(* IEC 61131-3 sources: com.logicals.lc3.webinar/usRTS_RPMControl_iSOC/src_FB_LIB_SAFE/Convert/LINT, 6 files *)

(* ---- wTRUNC_LINT_TO_DINT.iecst ---- *)
NAMESPACE logicals.web.standard
NAMESPACE convert

/*
 * Function block wrapper for IEC 61131-3 TO_DINT<br>
 * IN =  input value (LINT)<br>
 * OUT = IN (DINT)<br>
 */
FUNCTION_BLOCK wTRUNC_LINT_TO_DINT
	{ vNameAlignment:="center"; altName:="TRUNC_LINT_TO_DINT"; bgColor:="LightPink"; width:=180; hideIONames; }
	VAR_INPUT
		IN : LINT;
	END_VAR
	VAR_OUTPUT
		OUT: DINT;
	END_VAR

	OUT := TO_DINT(IN:=IN, ENO=>ENO);
END_FUNCTION_BLOCK

END_NAMESPACE
END_NAMESPACE

(* ---- wTRUNC_LINT_TO_INT.iecst ---- *)
NAMESPACE logicals.web.standard
NAMESPACE convert

/*
 * Function block wrapper for IEC 61131-3 TO_INT<br>
 * IN =  input value (LINT)<br>
 * OUT = IN (INT)<br>
 */
FUNCTION_BLOCK wTRUNC_LINT_TO_INT
	{ vNameAlignment:="center"; altName:="TRUNC_LINT_TO_INT"; bgColor:="LightPink"; width:=180; hideIONames; }
	VAR_INPUT
		IN : LINT;
	END_VAR
	VAR_OUTPUT
		OUT: INT;
	END_VAR

	OUT := TO_INT(IN:=IN, ENO=>ENO);
END_FUNCTION_BLOCK

END_NAMESPACE
END_NAMESPACE

(* ---- wTRUNC_LINT_TO_LREAL.iecst ---- *)
NAMESPACE logicals.web.standard
NAMESPACE convert

/*
 * Function block wrapper for IEC 61131-3 TO_LREAL<br>
 * IN =  input value (LINT)<br>
 * OUT = IN (LREAL)<br>
 */
FUNCTION_BLOCK wTRUNC_LINT_TO_LREAL
	{ vNameAlignment:="center"; altName:="TRUNC_LINT_TO_LREAL"; bgColor:="Orange"; width:=180; hideIONames; }
	VAR_INPUT
		IN : LINT;
	END_VAR
	VAR_OUTPUT
		OUT: LREAL;
	END_VAR

	OUT := TO_LREAL(IN:=IN, ENO=>ENO);
END_FUNCTION_BLOCK

END_NAMESPACE
END_NAMESPACE

(* ---- wTRUNC_LINT_TO_REAL.iecst ---- *)
NAMESPACE logicals.web.standard
NAMESPACE convert

/*
 * Function block wrapper for IEC 61131-3 TO_REAL<br>
 * IN =  input value (LINT)<br>
 * OUT = IN (REAL)<br>
 */
FUNCTION_BLOCK wTRUNC_LINT_TO_REAL
	{ vNameAlignment:="center"; altName:="TRUNC_LINT_TO_REAL"; bgColor:="Orange"; width:=180; hideIONames; }
	VAR_INPUT
		IN : LINT;
	END_VAR
	VAR_OUTPUT
		OUT: REAL;
	END_VAR

	OUT := TO_REAL(IN:=IN, ENO=>ENO);
END_FUNCTION_BLOCK

END_NAMESPACE
END_NAMESPACE

(* ---- wTRUNC_LINT_TO_SINT.iecst ---- *)
NAMESPACE logicals.web.standard
NAMESPACE convert

/*
 * Function block wrapper for IEC 61131-3 TO_SINT<br>
 * IN =  input value (LINT)<br>
 * OUT = IN (SINT)<br>
 */
FUNCTION_BLOCK wTRUNC_LINT_TO_SINT
	{ vNameAlignment:="center"; altName:="TRUNC_LINT_TO_SINT"; bgColor:="LightPink"; width:=180; hideIONames; }
	VAR_INPUT
		IN : LINT;
	END_VAR
	VAR_OUTPUT
		OUT: SINT;
	END_VAR

	OUT := TO_SINT(IN:=IN, ENO=>ENO);
END_FUNCTION_BLOCK

END_NAMESPACE
END_NAMESPACE

(* ---- wTRUNC_LINT_TO_ULINT.iecst ---- *)
NAMESPACE logicals.web.standard
NAMESPACE convert

/*
 * Function block wrapper for IEC 61131-3 TO_ULINT<br>
 * IN =  input value (LINT)<br>
 * OUT = IN (ULINT)<br>
 */
FUNCTION_BLOCK wTRUNC_LINT_TO_ULINT
	{ vNameAlignment:="center"; altName:="TRUNC_LINT_TO_ULINT"; bgColor:="Plum"; width:=180; hideIONames; }
	VAR_INPUT
		IN : LINT;
	END_VAR
	VAR_OUTPUT
		OUT: ULINT;
	END_VAR

	OUT := TO_ULINT(IN:=IN, ENO=>ENO);
END_FUNCTION_BLOCK

END_NAMESPACE
END_NAMESPACE
